Staubli VAL3: remGetJoints.pgx

program remGetJoints(string& sReturn[] (dimensions=1))
  local joint jPos
begin
  // Return the physical positions of the robot joints
  //
  logMsg("call remGetJoints")
  jPos=herej()
  sReturn="GETJOINTS"
  sReturn=sReturn+" "+toString(sNumConv,jPos.j1)
  sReturn=sReturn+" "+toString(sNumConv,jPos.j2)
  sReturn=sReturn+" "+toString(sNumConv,jPos.j3)
  sReturn=sReturn+" "+toString(sNumConv,jPos.j4)
  sReturn=sReturn+" "+toString(sNumConv,jPos.j5)
  sReturn=sReturn+" "+toString(sNumConv,jPos.j6)
end
